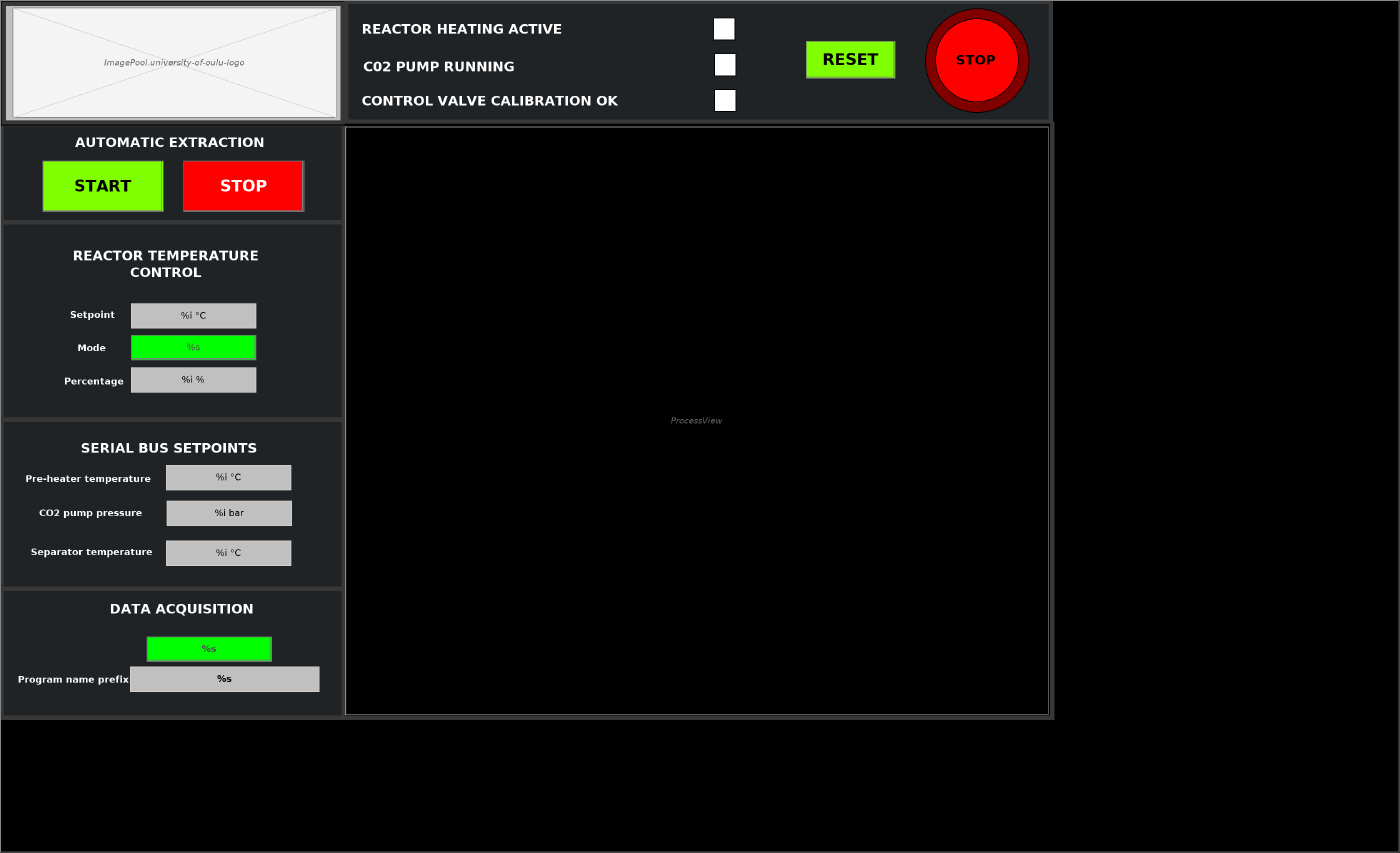
VISUALIZATION MainScreen_1_1  // 1680x1024
    Rectangle (413,0 850x148)
    Rectangle (2,151 411x709)
    Textfield (157,364 150x30), "%i °C", text variable: MainScreenBindings.ReactorTemperatureSetpointTextField_TextVariable
        OnMouseDown: write the text variable via VisuDialogs.Numpad, min 40, max 120
    Button (157,402 150x30), "%s", text variable: MainScreenBindings.RectorTemperatureControlModeButton_TextVariable, colour toggle: MainScreenBindings.PidParamMenuButton_Invisible
        toggle MainScreenBindings.RectorTemperatureControlModeButton_ToggleVariable
    Label (39,396 142x44), "Mode"
    Label (40,356 142x44), "Setpoint"
    Label (42,436 142x44), "Percentage", invisible if: MainScreenBindings.PercentageLabel_Invisible
    Textfield (157,441 150x30), "%i %", text variable: MainScreenBindings.ReactorTemperatureControlPercentageTextField_TextVariable, invisible if: MainScreenBindings.ReactorTemperatureControlPercentageTextField_Invisible
        OnMouseDown: write the text variable via VisuDialogs.Numpad, min 0, max 100
    Button (176,764 150x30), "%s", text variable: MainScreenBindings.StartMatlabButton_TextVariable, pressed state: RunMATLAB.bMatlabBtnState, input disabled if: MainScreenBindings.StartMatlabButton_DeactivateInputs
        p2175578022: MainScreenBindings.StartMatlabButton_Color
        toggle MainScreenBindings.StartMatlabButton_ToggleVariable
    Textfield (199,558 150x30), "%i °C", text variable: MainScreenBindings.PreHeaterTemperatureSetpointTextField_TextVariable
        OnMouseDown: write MainScreenBindings.PreHeaterTemperatureSetpointTextField_WriteAvariable via VisuDialogs.Numpad, min 0, max 120
    Label (35,553 142x44), "Pre-heater temperature"
    Textfield (200,601 150x30), "%i bar", text variable: MainScreenBindings.Co2PressureSetpointTextField_TextVariable
        OnMouseDown: write MainScreenBindings.Co2PressureSetpointTextField_WriteAvariable via VisuDialogs.Numpad, min 80, max 350
    Label (38,594 142x44), "CO2 pump pressure"
    Textfield (199,649 150x30), "%i °C", text variable: MainScreenBindings.SeparatorTemperatureSetpointTextField_TextVariable
        OnMouseDown: write MainScreenBindings.SeparatorTemperatureSetpointTextField_WriteAvariable via VisuDialogs.Numpad, min 0, max 100
    Label (39,641 142x44), "Separator temperature"
    Textfield (156,800 227x30), "%s", text variable: MainScreenBindings.ProgramNamePrefixTextField_TextVariable
        OnMouseDown: write the text variable via Edit
    Label (17,794 142x44), "Program name prefix"
    Button (51,193 145x61), "START", text variable: MainScreenBindings.ExtractiveOutOnOffValveButton_TextVariable, input disabled if: MainScreenBindings.StartAutomaticExtractionButton_DeactivateInputs
        toggle MainScreenBindings.StartAutomaticExtractionButton_ToggleVariable
    Rectangle (2,2 411x147)
    Image (15,9 389x132), image: ImagePool.university-of-oulu-logo
    Label (49,156 310x30), "AUTOMATIC EXTRACTION"
    Rectangle (410,151 5x713)
    Label (44,276 310x82), "REACTOR TEMPERATURE CONTROL"
    Label (2,497 402x82), "SERIAL BUS SETPOINTS"
    Label (63,690 310x82), "DATA ACQUISITION"
    Rectangle (-1,264 410x5)
    Rectangle (4,501 410x5)
    Rectangle (1,704 410x5)
    Rectangle (4,859 1261x5)
    Rectangle (-1,151 5x713)
    Ellipse (1110,10 125x125)
    Ellipse (1122,22 100x100), colour toggle: MainScreenBindings.StopButtonEllipse_ToggleColor
        tap MainScreenBindings.StopButtonEllipse_TapVariable
    Label (1113,55 116x34), "STOP"
    Label (433,65 283x30), "C02 PUMP RUNNING"
    Label (431,20 298x30), "REACTOR HEATING ACTIVE"
    RoundedRectangle (857,64 26x27), colour toggle: MainScreenBindings.Co2PumpRunningIndicatorRectangle_ToggleColor
    Label (431,106 360x30), "CONTROL VALVE CALIBRATION OK"
    RoundedRectangle (857,107 26x27), colour toggle: MainScreenBindings.CalibrationDoneIndicatorRectangle_ToggleColor
    RoundedRectangle (856,21 26x27), colour toggle: MainScreenBindings.ReactorHeatingActiveIndicatorRectangle_ToggleColor
    Button (220,193 145x61), "STOP", text variable: MainScreenBindings.ExtractiveOutOnOffValveButton_TextVariable, input disabled if: MainScreenBindings.StopAutomaticExtractionButton_DeactivateInputs
        toggle MainScreenBindings.StartAutomaticExtractionButton_ToggleVariable
    Rectangle (1260,146 5x713)
    Frame (414,152 844x706), invisible if: MainScreenBindings.ParameterViewFrame_Invisible, frame switch variable: MainScreenBindings.ProcessViewFrame_SwtichFrameVariable
        shows ProcessView()
        shows ParameterView()
    Button (967,49 107x45), "RESET", text variable: MainScreenBindings.ExtractiveOutOnOffValveButton_TextVariable, invisible if: MainScreenBindings.ResetButtonRectangle_Invisible
        tap MainScreenBindings.ResetButtonRectangle_TapVariable
        toggle MainScreenBindings.StartAutomaticExtractionButton_ToggleVariable
END_VISUALIZATION

(* stored: Version 1.1.0.1, ProductVersion 3.1.4024.9
   Visu MainScreen_1_1: Id {3e9d1ae6-676d-4aed-86fb-940379dd364b} *)
